FUNCTION F_NormSqVec3 : LREAL
VAR_INPUT
    iVec3 : I_Vec3;
END_VAR


F_NormSqVec3 := iVec3.x*iVec3.x + iVec3.y*iVec3.y + iVec3.z*iVec3.z;

END_FUNCTION

(* stored: Version 1.1.0.1
   POU F_NormSqVec3: Id {6c50c430-ce25-4aa8-8f5a-7d8b092b21bf}, SpecialFunc None *)
